FUNCTION_BLOCK FB_Lion IMPLEMENTS I_AnimalTraits
VAR_INPUT
END_VAR
VAR_OUTPUT
END_VAR
VAR
END_VAR

{warning 'add method implementation '}
METHOD DietType : BOOL
END_METHOD

{warning 'add method implementation '}
METHOD IsDangerous : BOOL
END_METHOD

END_FUNCTION_BLOCK

(* stored: Version 1.1.0.1, ProductVersion 3.1.4024.16
   POU FB_Lion: Id {b287a256-5f13-449a-a62a-1dbeb2582223}, SpecialFunc None
   Method DietType: Id {2427e0aa-09d4-4b85-a380-e88b200543b3}
   Method IsDangerous: Id {eb45f440-270d-4f48-9b81-bbf616392c05} *)
